FUNCTION_BLOCK FB_Supervisor
VAR_INPUT
	RemoteHost									 : T_IPv4Addr:='127.0.0.1';
	RemotePort									 : UDINT:=2000;
	CycleTime3002								 : TIME := T#100MS;
	CycleTime1026								 : TIME := T#30MS;
	Execute										 : BOOL; //Connect to Navitrol, and establish comuncations. If false, the socket is closed.
	st3002_Supervisor_Status					 : ST_3002_Supervisor_Status;
	st1026_Measurement_update_generic_omni_drive : ST_1026_Measurement_update_generic_omni_drive;
	Initialize_position							 : BOOL;//Rising edge trigger to send a Initialize position command
	st1001_Initialize_position					 : ST_1001_Initialize_position := (X := 100.0, Y := 150.0);
END_VAR

VAR_OUTPUT
	st3102_Navitrol_status			   : ST_3102_Navitrol_status;
	st1126_Motor_control_omni_response : ST_1126_Motor_control_omni_response;
	st1101_Position_initialized		   : ST_1101_Position_initialized;
	Busy							   : BOOL;
	Error							   : BOOL;
	ErrorID							   : UDINT;
END_VAR

VAR
	State : (INIT_FBs,
		CLOSE_OLD_SOCKETS,
		CONNECT_TO_Server,
		COMS_ACTIVE,
		CLOSE_CONNECTION);
	CloseAll							   : FB_SocketCloseAll;
	Connect								   : FB_SocketConnect;
	Timer3002							   : TON;
	Send3002							   : FB_SocketSend;
	Timer1026							   : TON;
	Send1026							   : FB_SocketSend;
	Close								   : FB_SocketClose;
	Receive								   : FB_SocketReceive;
	rtInitialize_position				   : R_TRIG;
	Send1001							   : FB_SocketSend;
	st1100_Position_initialization_started : ST_1100_Position_initialization_started;

	//Receive
	ReceiveBuffer			: U_Recived_bytes_from_Navitrol;
	NumOf1100MsgRecived		: UDINT;
	NumOf1101MsgRecived		: UDINT;	
	NumOf3102MsgRecived		: UDINT;
	NumOf1126MsgRecived		: UDINT;
	UnknowMsgRecivedCounter : UDINT;
	UnknowMsg				: U_Recived_bytes_from_Navitrol;

	//Event logging
	FirstScan  : BOOL := TRUE;
	ErrorMsg   : FB_TcMessage;
	VerboseMsg : FB_TcMessage;
END_VAR

IF FirstScan THEN
	ErrorMsg.CreateEx(stEventEntry := TC_EVENTS.TcpIpComms.ErrorMsg, ipSourceInfo := 0);
	VerboseMsg.CreateEx(stEventEntry := TC_EVENTS.TcpIpComms.VerboseMsg, ipSourceInfo := 0);
	FirstScan := FALSE;
END_IF

CASE State OF
	INIT_FBs: // Init State
		CloseAll(bExecute := FALSE);
		Connect(bExecute := FALSE);
		Send3002(bExecute := FALSE);
		Send1026(bExecute := FALSE);
		Receive(bExecute := FALSE);
		Close(bExecute := FALSE);
		Busy					:= FALSE;
		NumOf3102MsgRecived		:= 0;
		NumOf1126MsgRecived		:= 0;
		UnknowMsgRecivedCounter := 0;
		IF Execute THEN
			State := CLOSE_OLD_SOCKETS;
			Busy  := TRUE;
			Error := FALSE;
			VerboseMsg.ipArguments.Clear().AddString('Starting communications to:').AddString(RemoteHost).AddUDInt(RemotePort);
			VerboseMsg.Send();
		END_IF

	CLOSE_OLD_SOCKETS:
		CloseAll(sSrvNetId := '', bExecute := TRUE, tTimeout := T#10S);
		IF NOT CloseAll.bBusy THEN
			State := CONNECT_TO_Server;
		END_IF

	CONNECT_TO_Server:
		Connect(sSrvNetId	:= '',
				sRemoteHost := RemoteHost,
				nRemotePort := RemotePort,
				bExecute	:= TRUE,
				tTimeout	:= T#4S);

		IF Connect.hSocket.handle <> 0 AND NOT (Connect.bBusy) THEN
			State := COMS_ACTIVE;
			VerboseMsg.ipArguments.Clear().AddString('Connected to server:').AddString(RemoteHost).AddUDInt(RemotePort).AddString('Local port').AddUDInt(Connect.hSocket.localAddr.nPort);
			VerboseMsg.Send();
		ELSIF Connect.bError THEN
			Error := TRUE;
			State := INIT_FBs;
			ErrorMsg.ipArguments.Clear().AddString('Failed to connect to server:').AddString(RemoteHost).AddUDInt(RemotePort).AddString(', Error:').AddUDInt(Connect.nErrId);
			ErrorMsg.Send();
		END_IF

	COMS_ACTIVE:
		Timer3002(IN := NOT Timer3002.Q, PT := CycleTime3002);
		IF Timer3002.Q THEN
			st3002_Supervisor_Status.Protocol_version := 4;
			st3002_Supervisor_Status.Message_ID		  := 3002;
			st3002_Supervisor_Status.Message_length	  := SIZEOF(st3002_Supervisor_Status);
		END_IF

		Send3002(sSrvNetId := '',
				 hSocket   := Connect.hSocket,
				 cbLen	   := SIZEOF(st3002_Supervisor_Status),
				 pSrc	   := ADR(st3002_Supervisor_Status),
				 bExecute  := Timer3002.Q,
				 tTimeout  := T#2S);

		IF Send3002.bError THEN
			ErrorMsg.ipArguments.Clear().AddString('Failed to send 3002 Error:').AddUDInt(Send3002.nErrId);
			ErrorMsg.Send();
			State	:= CLOSE_CONNECTION;
			Error	:= TRUE;
			ErrorID := Send3002.nErrId;
		END_IF

		Timer1026(IN := NOT Timer1026.Q, PT := CycleTime1026);
		IF Timer1026.Q THEN
			st1026_Measurement_update_generic_omni_drive.Protocol_version := 4;
			st1026_Measurement_update_generic_omni_drive.Message_ID		  := 1026;
			st1026_Measurement_update_generic_omni_drive.Message_length	  := SIZEOF(st1026_Measurement_update_generic_omni_drive);
			st1026_Measurement_update_generic_omni_drive.Message_number	  := st1026_Measurement_update_generic_omni_drive.Message_number + 1;
		END_IF

		Send1026(sSrvNetId := '',
				 hSocket   := Connect.hSocket,
				 cbLen	   := SIZEOF(st1026_Measurement_update_generic_omni_drive),
				 pSrc	   := ADR(st1026_Measurement_update_generic_omni_drive),
				 bExecute  := Timer1026.Q,
				 tTimeout  := T#2S);

		IF Send1026.bError THEN
			ErrorMsg.ipArguments.Clear().AddString('Failed to send 1026 Error:').AddUDInt(Send1026.nErrId);
			ErrorMsg.Send();
			State	:= CLOSE_CONNECTION;
			Error	:= TRUE;
			ErrorID := Send1026.nErrId;
		END_IF

		rtInitialize_position(CLK := Initialize_position);
		IF rtInitialize_position.Q THEN
			st1001_Initialize_position.Protocol_version := 4;
			st1001_Initialize_position.Message_ID		:= 1001;
			st1001_Initialize_position.Message_length	:= SIZEOF(st1001_Initialize_position);
			MEMSET(destAddr:=ADR(st1101_Position_initialized),fillByte:=0,n:=SIZEOF(st1101_Position_initialized));
		END_IF

		Send1001(sSrvNetId := '',
				 hSocket   := Connect.hSocket,
				 cbLen	   := SIZEOF(st1001_Initialize_position),
				 pSrc	   := ADR(st1001_Initialize_position),
				 bExecute  := rtInitialize_position.Q,
				 tTimeout  := T#2S);

		IF Send1001.bError THEN
			ErrorMsg.ipArguments.Clear().AddString('Failed to send 1001 Error:').AddUDInt(Send1001.nErrId);
			ErrorMsg.Send();
		END_IF

		Receive(sSrvNetId := '',
				hSocket	  := Connect.hSocket,
				cbLen	  := SIZEOF(ReceiveBuffer),
				pDest	  := ADR(ReceiveBuffer),
				bExecute  := TRUE,
				tTimeout  := T#10S);

		IF NOT Receive.bBusy THEN
			IF Receive.nRecBytes <> 0 THEN
				CASE ReceiveBuffer.Header.Message_ID OF //Check what message type is being recived - then copy it into the correct structure
					1100:
						NumOf1100MsgRecived := NumOf1100MsgRecived + 1;
						MEMCPY(destAddr := ADR(st1100_Position_initialization_started), srcAddr := ADR(ReceiveBuffer), n := SIZEOF(st1100_Position_initialization_started));
						VerboseMsg.ipArguments.Clear().AddString('Position initialization started');
						VerboseMsg.Send();
					1101:
						NumOf1101MsgRecived := NumOf1101MsgRecived + 1;
						MEMCPY(destAddr := ADR(st1101_Position_initialized), srcAddr := ADR(ReceiveBuffer), n := SIZEOF(st1101_Position_initialized));
						VerboseMsg.ipArguments.Clear().AddString('Position initialization finished');
						VerboseMsg.Send();

					1126:
						NumOf1126MsgRecived := NumOf1126MsgRecived + 1;
						MEMCPY(destAddr := ADR(st1126_Motor_control_omni_response), srcAddr := ADR(ReceiveBuffer), n := SIZEOF(st1126_Motor_control_omni_response));

					3102:
						NumOf3102MsgRecived := NumOf3102MsgRecived + 1;
						MEMCPY(destAddr := ADR(st3102_Navitrol_status), srcAddr := ADR(ReceiveBuffer), n := SIZEOF(st3102_Navitrol_status));

				ELSE
					UnknowMsgRecivedCounter := UnknowMsgRecivedCounter + 1;
					MEMCPY(destAddr := ADR(UnknowMsg), srcAddr := ADR(ReceiveBuffer), n := SIZEOF(UnknowMsg));
					ErrorMsg.ipArguments.Clear().AddString('Unknow msg type recived with ID:').AddUInt(ReceiveBuffer.Header.Message_ID);
					ErrorMsg.Send();
				END_CASE
			END_IF

			Receive(bExecute := FALSE);

			//Clear recive buffer
			MEMSET(destAddr := ADR(ReceiveBuffer), fillByte := 0, n := SIZEOF(ReceiveBuffer));
		END_IF

		IF Receive.bError THEN
			ErrorMsg.ipArguments.Clear().AddString('Failed to Receive Error:').AddUDInt(Receive.nErrId);
			ErrorMsg.Send();
			State	:= CLOSE_CONNECTION;
			Error	:= TRUE;
			ErrorID := Receive.nErrId;
		END_IF

		IF NOT Execute THEN
			VerboseMsg.ipArguments.Clear().AddString('Connection closed by user');
			VerboseMsg.Send();
			State := CLOSE_CONNECTION;
		END_IF

	CLOSE_CONNECTION:
		Close( // Close connection
			sSrvNetId := '',
			hSocket	  := Connect.hSocket,
			bExecute  := TRUE,
			tTimeout  := T#4S);

		IF NOT Close.bBusy THEN
			Close(bExecute := FALSE);
			State := INIT_FBs;
		END_IF
END_CASE

END_FUNCTION_BLOCK

(* stored: Version 1.1.0.1, ProductVersion 3.1.4026.17
   POU FB_Supervisor: Id {ba3b2abf-990a-4014-84c0-14af22135bdc}, SpecialFunc None *)
